Fanuc KAREL source: kt00478.KL

PROGRAM KT00478
%STACKSIZE=65535
%PRIORITY=65535
%NOLOCKGROUP
VAR
P1 : POSITION
P2 : XYZWPR
OUT : BOOLEAN
BEGIN
P2.Y=2.0
-- UNRESOLVED_PC line 9 opcodes [49 49 7E AC 23] marker_code=20
END KT00478
